FUNCTION_BLOCK FB_MotionInterlocksCommon_TestDouble IMPLEMENTS I_MotionInterlocksCommon
VAR
    bPowerEnabled: BOOL:=FALSE;
   // NC STO Input: TRUE if ok to move
    bHardwareEnable : BOOL ;
    bUserEnable: BOOL := TRUE;
    bEnable: BOOL;
    bReset : BOOL;
    sMessage : STRING;
    bError : BOOL;
    nErrorID : UDINT;
    // Set by default, an error condition will reset this
    bMoveOk : BOOL := TRUE;

END_VAR

METHOD DriveCommands
VAR_INPUT
    MoveEnable: BOOL;
    NewMoveReq : BOOL;
END_VAR
THIS^.bEnable := MoveEnable;
END_METHOD

{warning 'Add method implementation '}
METHOD EnableInterlocks
VAR_INPUT
	UserEnable	: BOOL;
	HardwareEnable	: BOOL;
END_VAR
END_METHOD

PROPERTY Error : BOOL
GET
Error := bError;
END_GET
SET
bError := Error;
END_SET
END_PROPERTY

PROPERTY ErrorID : UDINT
GET
ErrorID := nErrorID;
END_GET
SET
nErrorID := ErrorID;
END_SET
END_PROPERTY

PROPERTY HardwareEnable : BOOL
GET
END_GET
SET
bHardwareEnable := HardwareEnable;
END_SET
END_PROPERTY

PROPERTY Message : T_MAXSTRING
GET
Message := sMessage;
END_GET
SET
sMessage := Message;
END_SET
END_PROPERTY

PROPERTY MoveOk : BOOL
GET
MoveOk := bMoveOk;
END_GET
SET
END_SET
END_PROPERTY

PROPERTY PowerEnabled : BOOL
GET
PowerEnabled :=bPowerEnabled;
END_GET
SET
END_SET
END_PROPERTY

METHOD Reset
END_METHOD

METHOD ResetErrors
VAR_INPUT
END_VAR
bError := FALSE;
nErrorID:= 0;
sMessage:='';
END_METHOD

PROPERTY UserEnable : BOOL
GET
END_GET
SET
bUserEnable := UserEnable;
END_SET
END_PROPERTY

END_FUNCTION_BLOCK

(* stored: Version 1.1.0.1
   POU FB_MotionInterlocksCommon_TestDouble: Id {0e1c2779-867c-4949-8b00-00663dc282f6}, SpecialFunc None
   Method DriveCommands: Id {01a235bb-6a8d-4b51-8c0a-3d8136ab49a6}
   Method EnableInterlocks: Id {55d66cb8-994d-4b8e-b57a-3c76e5fb91ea}
   Property Error: Id {68ade204-75fc-4d54-adb8-ed5abf657582}
   Get Get: Id {f1934e38-0a7e-47f5-9782-5973b0818453}
   Set Set: Id {d41f6317-6d37-4c46-8c7c-2e1ee780d122}
   Property ErrorID: Id {6ab6af77-b85e-4d3a-a1c5-a28baa23967c}
   Get Get: Id {b8d97dab-8e94-4574-a6de-28883ff7eca3}
   Set Set: Id {496fd04b-6a6f-45d3-8611-0cd595ec417b}
   Property HardwareEnable: Id {b61e843a-e16f-4bf9-a751-e2ee9ca06f64}
   Get Get: Id {198c931d-a063-4af8-8ab2-5c27a9ebe0d5}
   Set Set: Id {d2f9e458-e833-43c5-9f95-fd2c6475a0fd}
   Property Message: Id {fb98df5d-fd1f-44f8-a156-a62ef268f09b}
   Get Get: Id {98cdbec5-2a77-434d-917c-50ee0e45ed7d}
   Set Set: Id {56003863-6094-41be-8870-2fd02e9f9b1e}
   Property MoveOk: Id {567a542a-8bff-430c-bb26-a30f927d8d8a}
   Get Get: Id {bd01effb-06eb-4d8c-a796-aa7890a0db64}
   Set Set: Id {5f738456-0381-45f9-8495-6f474b182629}
   Property PowerEnabled: Id {c3ce75de-aded-4122-b66c-ef67e08fdb8d}
   Get Get: Id {edb6f6ad-751d-422f-8834-d24703acdb9e}
   Set Set: Id {6564c5fa-a989-44af-8901-719e1b37e561}
   Method Reset: Id {45939870-a895-412f-94d4-338002dacd8f}
   Method ResetErrors: Id {f36f7e3b-4b1e-4387-89e2-e52b4f418e83}
   Property UserEnable: Id {b67c8bc2-c5d8-44a8-a2c7-8252c58bf9ac}
   Get Get: Id {222086fa-1659-43ab-aa5a-6b671d1bafd5}
   Set Set: Id {d6a210bb-b3eb-46b0-93df-85780ce3e949} *)
